FUNCTION_BLOCK SUB_TIME_TIME (* a simple FB Function Block Type *)
  (* Standard: 61499-1; Type: Simple FB; Description: Template for a Simple FB *)
  (* Version 0.2, 2020-05-24, JHC, Holobloc Inc, Added ECC documentation. *)
  (* Version 0.1, 2020-05-19, JHC, Holobloc Inc, Changed name from SimpleFB back to Simple. *)
  (* Version 0.0, 2020-05-05, JHC, Holobloc Inc *)
  PACKAGE fb.rt.DIAS;
  IMPORT fb.datatype.*;
  IMPORT fb.rt.*;
  (* Compiler Java AdoptOpenJDK JDK 1.8.0_222 *)
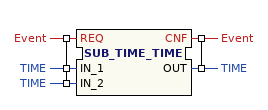
  EVENT_INPUT
    REQ WITH IN_1, IN_2; (* Service Request *)
  END_EVENT
  EVENT_OUTPUT
    CNF WITH OUT; (* Confirmation of Requested Service *)
  END_EVENT
  VAR_INPUT
    IN_1 : TIME; (* Input Variable *)
    IN_2 : TIME;
  END_VAR
  VAR_OUTPUT
    OUT : TIME; (* Output variable *)
  END_VAR
  VAR
    MULT : INT := 1;
  END_VAR
  EC_STATES
    REQ : REQ -> CNF; (* Services REQ event *)
  END_STATES
  ALGORITHM REQ IN ST: (* Normally Executed Algorithm *)
OUT := IN_1 - MULT*IN_2;
MULT := MULT + 1;
  END_ALGORITHM
END_FUNCTION_BLOCK
